TYPE ST_HMI_GRID_IN :
STRUCT
	nSelectedRowIndex	: UINT;
	nSelectedColumIndex	: UINT;	
END_STRUCT
END_TYPE

(* stored: Version 1.1.0.1
   DUT ST_HMI_GRID_IN: Id {82efbb16-4c1f-4654-bb5c-9dadfc7cae89} *)
